{attribute addProperty BoxType "EK1100-0000-0018"}
{attribute addProperty Id "Beckhoff_CUxxxxEK1122Beckhoff_CUxxxxEK1122_8084EAF6966120.75"}
{attribute addProperty CRC "3581622821"}
{attribute addProperty SizeInBites "966"}
{attribute addProperty SizeInBytes "120.75"}
TYPE Beckhoff_CUxxxx_D57B3A25 EXTENDS EK1100_179A0949 :
STRUCT
	{attribute addProperty Name "Beckhoff_CUxxxxEK1122"}
	Beckhoff_CUxxxxEK1122 : Beckhoff_CUxxxxEK1122_8084EAF6;
END_STRUCT
END_TYPE

(* stored: Version 1.2.0.0, ProductVersion 3.1.4024.9
   DUT Beckhoff_CUxxxx_D57B3A25: Id {bbc68efb-501c-411d-838e-898b088dbe94} *)
